TYPE M3RotationTargetStatuses :
STRUCT
	targetStatus: M3TargetStatus;
END_STRUCT
END_TYPE

(* stored: Version 1.1.0.1, ProductVersion 3.1.4019.2
   DUT M3RotationTargetStatuses: Id {e27f671f-a44f-409e-a47c-ca441a111e44} *)
